// SIMATIC STEP 7 (V5.x) project From_A_to_B
// CPU: CPU315-2 PN/DP(1)
// station: P_ADR_BUS
// station: Hardware
// station: SIMATIC 300
// program: S7 Program(1)

SYMBOL_TABLE
"Sensor_At_B"	I 0.0	BOOL	// Sensor de presença no ponto B
"Start_Button"	I 0.1	BOOL	// Botão para iniciar o processo
"Cycle Execution"	OB 1	OB 1
"Conveyor_Motor"	Q 0.0	BOOL	// Motor da esteira transportadora
END_SYMBOL_TABLE

ORGANIZATION_BLOCK "Cycle Execution"	// OB 1
TITLE = "Main Program Sweep (Cycle)"
VERSION : 0.1
VAR_TEMP
  OB1_EV_CLASS : BYTE ;	//Bits 0-3 = 1 (Coming event), Bits 4-7 = 1 (Event class 1)
  OB1_SCAN_1 : BYTE ;	//1 (Cold restart scan 1 of OB 1), 3 (Scan 2-n of OB 1)
  OB1_PRIORITY : BYTE ;	//Priority of OB Execution
  OB1_OB_NUMBR : BYTE ;	//1 (Organization block 1, OB1)
  OB1_RESERVED_1 : BYTE ;	//Reserved for system
  OB1_RESERVED_2 : BYTE ;	//Reserved for system
  OB1_PREV_CYCLE : INT ;	//Cycle time of previous OB1 scan (milliseconds)
  OB1_MIN_CYCLE : INT ;	//Minimum cycle time of OB1 (milliseconds)
  OB1_MAX_CYCLE : INT ;	//Maximum cycle time of OB1 (milliseconds)
  OB1_DATE_TIME : DATE_AND_TIME ;	//Date and time OB1 started
END_VAR
BEGIN
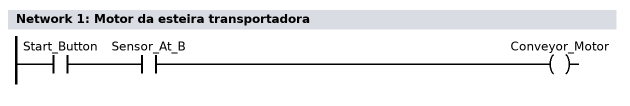
NETWORK
TITLE = Motor da esteira transportadora
      A     "Start_Button";
      A     "Sensor_At_B";
      =     "Conveyor_Motor";
END_ORGANIZATION_BLOCK
